{attribute 'call_after_init'}
FUNCTION_BLOCK FB_IOMappingJson EXTENDS FB_JsonSchemaEx_OLD
VAR_OUTPUT
	P_sJsonid			: MPM_JsonParser.DUT_JsonSchema := (member := '_id', typeClass := E_TypeClassEx.TYPE_STRING,jsonValueRoot := jsonRoot);
	P_sJsonTimeStamp	: MPM_JsonParser.DUT_JsonSchema := (member := 'time_stamp', typeClass := E_TypeClassEx.TYPE_FILETIME,jsonValueRoot := jsonRoot);		
	P_sJsonValues		: MPM_JsonParser.DUT_JsonSchema := (member := 'values', typeClass := E_TypeClassEx.TYPE_JSON,jsonValueRoot := jsonRoot);
END_VAR
VAR
	jsonRoot : SJsonValue;	
END_VAR
VAR_OUTPUT
	//stIOMappingEthercat : ARRAY [0..NUM_OF_VARS] OF ST_IOMappingEthercatJson;	
END_VAR
VAR CONSTANT
	//NUM_OF_VARS : DINT := -1 + (SIZEOF(ST_Vars_IO_Mapping_Ethercat)/8) ;// 8 is SIZEOF(PVOID) (SIZEOF(ST_IO_Mapping)/SIZEOF(PVOID)) -1 won't complie
END_VAR

METHOD INTERNAL M_Add1 : UDINT
VAR_INPUT
	x : REFERENCE TO UDINT;
END_VAR
M_Add1 := x;
x := x + 1;
END_METHOD

METHOD PUBLIC  M_CreateSchemaJson : BOOL
VAR_IN_OUT
END_VAR
VAR
	json : sJsonValue;
END_VAR
jsonRoot := THIS^.NewDocument();
M_SetJsonSchema(jsonRoot,P_sJsonid);
//M_SetJsonSchema(P_sJsonid.jsonValue,P_sJsonRecipe);
M_SetJsonSchema(jsonRoot,P_sJsonValues);
M_SetJsonSchema(jsonRoot,P_sJsonTimeStamp);
END_METHOD

METHOD PUBLIC M_GetIOMappingJson : HRESULT
VAR_INPUT
	lastResult : HRESULT;
END_VAR
VAR_INPUT
	path : STRING;
END_VAR
VAR_IN_OUT
	stIOMapping : ARRAY [*] OF ST_IOMappingJson;
END_VAR
VAR_INPUT
	fbIOMapping : POINTER TO FB_IOMapping;	
END_VAR
VAR
	pJson : SJsonValue;
	upperBound : DINT; 
END_VAR
VAR_INST
	loadFile : BOOL;		
	x : UDINT;
	fileName : STRING;
	_state			: DINT;
	_fbResult		: FB_ResultHelper;	
	errorCode : HRESULT;
END_VAR
//THIS^.CopyDocument(aStringJson,SIZEOF(aStringJson));

IF _fbResult.M_MethodResult(M_GetIOMappingJson,lastResult) = FALSE THEN
	RETURN;
ELSE
	
	IF _fbResult.P_Result = E_Result.S_OK THEN //Reset
		_state := 0;	
		x := 0;
		fileName := path;
		loadFile := FALSE;
		THIS^.LoadDocumentFromFile(fileName,loadFile,hrErrorCode => errorCode);
		loadFile := TRUE;
	END_IF 
	
	_fbResult.P_Result := E_Result.S_WORKING; //Working	
	
	CASE _state OF
		0:	
			THIS^.LoadDocumentFromFile(fileName,loadFile,hrErrorCode => errorCode);
			IF loadFile = FALSE AND errorCode = 0 THEN
				_state := 1;
			ELSIF loadFile = FALSE AND errorCode < 0 THEN
				_fbResult.P_Result := E_Result.S_FAILED; //Working	
			END_IF		
		1:
			THIS^.M_PraseSchemaJson();
			upperBound := UPPER_BOUND(stIOMapping,1);
			FOR x := 0 TO upperBound BY 1 DO
				pJson := THIS^.FindMember(P_sJsonValues.jsonValue,stIOMapping[x].name);	
				IF pJson > 0 THEN
					THIS^.M_GetIOMappingJson_Values(pJson,ADR(stIOMapping[x]),fbIOMapping);
				END_IF	
			END_FOR
			_fbResult.P_Result := E_Result.S_OK; //Working
	END_CASE	

END_IF
END_METHOD

METHOD PROTECTED M_GetIOMappingJson_Values : HRESULT
VAR_INPUT
	pJson : SJsonValue;
	stIOMapping : POINTER TO ST_IOMappingJson;	
	fbIOMapping : POINTER TO FB_IOMapping;
END_VAR
VAR
END_VAR
THIS^.M_GetJsonMemberValue(pJson,'deviceNum',stIOMapping^.deviceNum);
THIS^.M_GetJsonMemberValue(pJson,'channel',stIOMapping^.channel);

THIS^.M_GetJsonMemberValue(pJson,'ethercatDeviceNum',stIOMapping^.ethercatDeviceNum);
THIS^.M_GetJsonMemberValue(pJson,'ioLinkDevice',stIOMapping^.ioLinkDevice);
THIS^.M_GetJsonMemberValue(pJson,'ioLinkSlaveChannel',stIOMapping^.ioLinkSlaveChannel);


IF stIOMapping^.deviceNum > 0 AND_THEN fbIOMapping^.ip.M_GetRef_PVOID((stIOMapping^.pAny.pvalue),stIOMapping^.deviceNum,stIOMapping^.channel) = MPM_FBResult.E_Result.S_FAILED THEN
	M_GetIOMappingJson_Values := E_Result.S_FAILED;
ELSIF stIOMapping^.ethercatDeviceNum > 0 AND_THEN fbIOMapping^.ip.M_GetRefIOLink_PVOID((stIOMapping^.pAny.pvalue),stIOMapping^.ethercatDeviceNum,stIOMapping^.ioLinkDevice,stIOMapping^.ioLinkSlaveChannel) = MPM_FBResult.E_Result.S_FAILED THEN
	M_GetIOMappingJson_Values :=  E_Result.S_FAILED;;	
END_IF

M_GetIOMappingJson_Values :=  E_Result.S_OK;
END_METHOD

METHOD PUBLIC  M_PraseSchemaJson : BOOL
VAR_INPUT
END_VAR
VAR
END_VAR
jsonRoot := THIS^.GetDocumentRoot();
IF jsonRoot > 0 THEN
	M_PraseJsonSchema(jsonRoot,P_sJsonid);
	//M_SetJsonSchema(P_sJsonid.jsonValue,P_sJsonRecipe);
	M_PraseJsonSchema(jsonRoot,P_sJsonValues);
	M_PraseJsonSchema(jsonRoot,P_sJsonTimeStamp);
END_IF
END_METHOD

METHOD PUBLIC M_SetIOMappingJson : HResult
VAR_INPUT
	lastResult : HRESULT;
END_VAR
VAR_INPUT
	path : STRING(255);
END_VAR
VAR_IN_OUT
	stIOMapping : ARRAY [*] OF ST_IOMappingJson;
END_VAR
VAR
	pJson : SJsonValue;
	upperBound : DINT; 
END_VAR
VAR_INST
	saveFile : BOOL;		
	x : UDINT;
	fileName : STRING(255);
	_state			: DINT;
	_fbResult		: FB_ResultHelper;	
	errorCode : HRESULT;
END_VAR
IF _fbResult.M_MethodResult(M_SetIOMappingJson,lastResult) = FALSE THEN
	RETURN;
ELSE
	
	IF _fbResult.P_Result = E_Result.S_OK THEN //Reset
		_state := 0;	
		x := 0;
		fileName := path;
		saveFile := FALSE;
		THIS^.SaveDocumentToFile(fileName,saveFile,hrErrorCode => errorCode);
		saveFile := TRUE;
	END_IF 
	
	_fbResult.P_Result := E_Result.S_WORKING; //Working	
	
	CASE _state OF
		0:	
			upperBound := UPPER_BOUND(stIOMapping,1);
			THIS^.M_CreateSchemaJson();
			
			FOR x := 0 TO upperBound BY 1 DO
				pJson := THIS^.M_SetJsonMember(P_sJsonValues.jsonValue,stIOMapping[x].name);		(* 3 Inches *)			
				THIS^.M_SetIOMappingJson_Values(pJson);
			END_FOR
			
			_state := 1;
		1:	
			THIS^.SaveDocumentToFile(fileName,saveFile,hrErrorCode => errorCode);
			IF saveFile = FALSE AND errorCode = 0 THEN
				_fbResult.P_Result := E_Result.S_OK; //Working	
			ELSIF saveFile = FALSE AND errorCode < 0 THEN
				_fbResult.P_Result := E_Result.S_FAILED; //Working	
			END_IF		
	END_CASE		
END_IF	



(*


*)
END_METHOD

METHOD PROTECTED M_SetIOMappingJson_Values : BOOL
VAR_INPUT
	pJson : SJsonValue;
END_VAR
VAR
	stIOMapping : ST_IOMappingJson;
END_VAR
THIS^.M_SetJsonMemberValue(pJson,'deviceNum',stIOMapping.deviceNum);
THIS^.M_SetJsonMemberValue(pJson,'channel',stIOMapping.channel);

THIS^.M_SetJsonMemberValue(pJson,'ethercatDeviceNum',stIOMapping.ethercatDeviceNum);
THIS^.M_SetJsonMemberValue(pJson,'ioLinkDevice',stIOMapping.ioLinkDevice);
THIS^.M_SetJsonMemberValue(pJson,'ioLinkSlaveChannel',stIOMapping.ioLinkSlaveChannel);
END_METHOD

END_FUNCTION_BLOCK

(* stored: Version 1.1.0.1, ProductVersion 3.1.4024.12
   POU FB_IOMappingJson: Id {968e0526-87bd-43a3-9481-27cbde56a774}, SpecialFunc None
   Folder Protected: Id {b763cb27-a438-4539-88cf-8606754f6eb0}
   Method M_Add1: Id {dbabb5bf-50a4-4da3-bb26-04dfb18d71d3}
   Method M_CreateSchemaJson: Id {3c46d5e4-1d88-47c1-8fab-14a7ed2c9fdc}
   Method M_GetIOMappingJson: Id {e3d0a72b-79c2-4ef9-9f9e-050402784e03}
   Method M_GetIOMappingJson_Values: Id {25fa4365-bd8e-4b91-b974-56469712982f}
   Method M_PraseSchemaJson: Id {6d4af479-2ba9-44db-b820-4b91b6a16946}
   Method M_SetIOMappingJson: Id {b9332636-1be0-465b-a801-3c6bee232a52}
   Method M_SetIOMappingJson_Values: Id {d0eac7ea-4c8d-4908-9165-e7764edfc234} *)
